% RSLogix 500 project MCR_Class.RSS, saved by version 8.30.00.16 %
PROJECT "UNTITLED"    % processor: MicroLogix 1000 %

PROGRAM FILES
  LAD 2 "MAIN_PROG"  13 rungs
  LAD 3 "USER_FAULT"  1 rungs
  LAD 4 "HSC_INT"  1 rungs
  LAD 5 "STI_INT"  1 rungs
  LAD 6, 7, 8, 9, 10, 11, 12, 13, 14, 15, 16: only END

DATA FILES
  O0 OUTPUT  1 elements
  I1 INPUT  2 elements
  S2 STATUS  33 elements
  B3 BINARY  32 elements
  T4 TIMER  40 elements
  C5 COUNTER  32 elements
  R6 CONTROL  16 elements
  N7 INTEGER  105 elements

LADDER 2 "MAIN_PROG"
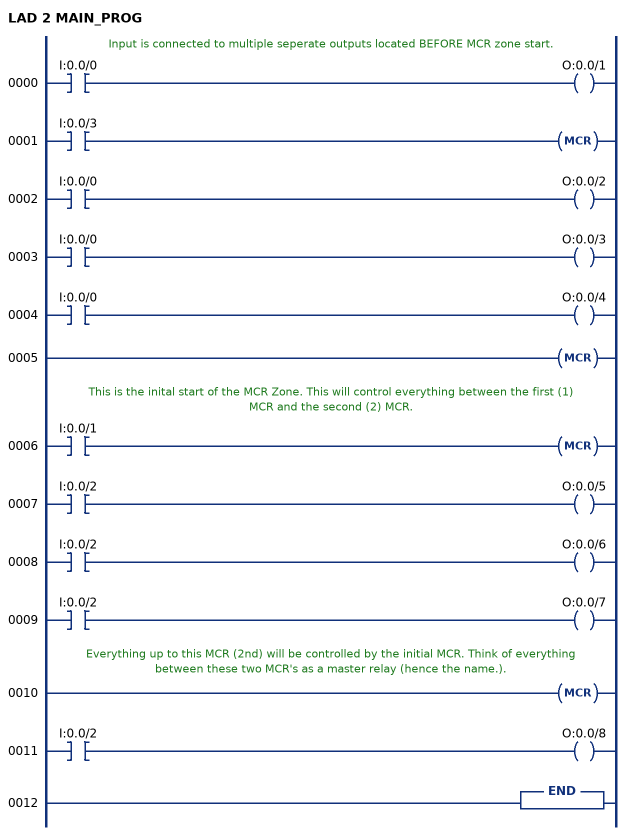
% Rung: 0 %
% Input is connected to multiple seperate outputs located BEFORE MCR zone start. %
SOR XIC I:0.0/0 OTE O:0.0/1 EOR
% Rung: 1 %
SOR XIC I:0.0/3 MCR EOR
% Rung: 2 %
SOR XIC I:0.0/0 OTE O:0.0/2 EOR
% Rung: 3 %
SOR XIC I:0.0/0 OTE O:0.0/3 EOR
% Rung: 4 %
SOR XIC I:0.0/0 OTE O:0.0/4 EOR
% Rung: 5 %
SOR MCR EOR
% Rung: 6 %
% This is the inital start of the MCR Zone. This will control everything between the first (1) MCR and the second (2) MCR. %
SOR XIC I:0.0/1 MCR EOR
% Rung: 7 %
SOR XIC I:0.0/2 OTE O:0.0/5 EOR
% Rung: 8 %
SOR XIC I:0.0/2 OTE O:0.0/6 EOR
% Rung: 9 %
SOR XIC I:0.0/2 OTE O:0.0/7 EOR
% Rung: 10 %
% Everything up to this MCR (2nd) will be controlled by the initial MCR. Think of everything between these two MCR's as a master relay (hence the name.). %
SOR MCR EOR
% Rung: 11 %
SOR XIC I:0.0/2 OTE O:0.0/8 EOR
% Rung: 12 %
SOR END EOR

REVISION NOTES
  0: Added comments to clarify function.
